{attribute 'qualified_only'}
{attribute 'strict'}
{attribute 'to_string'}
TYPE E_EventType :
(
    Verbose  := 0, 
    Info     := 1, 
    Warning  := 2, 
    Error    := 3, 
    Critical := 4
);
END_TYPE

(* stored: Version 1.1.0.1, ProductVersion 3.1.4024.15
   EnumerationTextList E_EventType: Id {cfebfd1b-e071-4b13-88ae-81f3d3e85ed8} *)
